# EPICS substitutions: iocs/hexapod-demo/hexapodDemoApp/Db/hexapodDemo_expanded.substitutions
# This file was automatically generated on Thu 15 Nov 2018 14:28:58 GMT from
# source: /home/hgv27681/R3.14.12.7/support/pmac/etc/makeIocs/lab.xml
#
# *** Please do not edit this file: edit the source file instead. ***
#

# Macros:
#  PORT      The asyn port for the pmac controller
#  P         PV Prefix
#  R         PV Device
file $(SYMETRIE)/db/SymetriePmac.template
{
pattern { PORT, P, R }
    { "HEXAPOD", "SYM", ":HEX01:" }
}
